// TIA Portal V20 export
DATA_BLOCK "BK13"   // DB282
// stored: MemoryReserve 100
   VAR
      "X10-1.CATHODE ALIGN TABLE Y1-AXIS LIMIT SENSOR(-)" : Bool := TRUE;
      "X11-1.CATHODE ALIGN TABLE Y1-AXIS LIMIT SENSOR(+)" : Bool := TRUE;
      "X12-1.CATHODE ALIGN TABLE X-AXIS LIMIT SENSOR(-)" : Bool := TRUE;
      "X13-1.CATHODE ALIGN TABLE X-AXIS LIMIT SENSOR(+)" : Bool := TRUE;
      "X14-1.CATHODE ALIGN TABLE Y2-AXIS LIMIT SENSOR(-)" : Bool := TRUE;
      "X15-1.CATHODE ALIGN TABLE Y2-AXIS LIMIT SENSOR(+)" : Bool := TRUE;
      "X16-1.CATHODE ALIGN TABLE ELECTRODE DETECT SENSOR" : Bool := FALSE;
      "X17-1.CATHODE ALIGN TABLE PRESSURE SWITCH" : Bool := FALSE;
      "X10-2.CATHODE ALIGN TABLE Y1-AXIS HOME SENSOR" : Bool := TRUE;
      "X11-2.SPARE" : Bool := FALSE;
      "X12-2.CATHODE ALIGN TABLE X-AXIS HOME SENSOR" : Bool := FALSE;
      "X13-2.SPARE" : Bool := FALSE;
      "X14-2.CATHODE ALIGN TABLE Y2-AXIS HOME SENSOR" : Bool := FALSE;
      "X15-2.SPARE" : Bool := FALSE;
      "X16-2.SPARE" : Bool := FALSE;
      "X17-2.SPARE" : Bool := FALSE;
   END_VAR
BEGIN
END_DATA_BLOCK
